	// Increment component byte offset
	offset := offset + SIZEOF(ST_RTComponentData) + qrtComponent[comp].nSize;
END_FOR

// Get hook position
IF bActive THEN
	IF markerComponent.nMarkers >= 2 THEN
		// Reset eMin to a default "high" value
		eMin := 1E10;
		
		FOR i := 0 TO markerComponent.nMarkers DO
			FOR j := 0 TO markerComponent.nMarkers DO
				// Calculate norm
				d := GetNorm(markerComponent.markers[i], markerComponent.markers[j]);
				e := ABS(d - dMarker);
				
				// Check if current marker set is closer than the others
				IF e < eMin THEN
					eMin := e;
					
					dSave := d;
					iSave := i;
					jSave := j;
				END_IF
			END_FOR
		END_FOR
		// Pick saved markers
		iMarker := markerComponent.markers[iSave];
		jMarker := markerComponent.markers[jSave];
		
		// Calculate average marker
		feedback.dist := dSave/1000.0;
		
		xSave := (iMarker.x + jMarker.x)/2.0;
		ySave := (iMarker.y + jMarker.y)/2.0;
		zSave := (iMarker.z + jMarker.z)/2.0;
		
	ELSIF markerComponent.nMarkers = 1 THEN
		// Indicate that hook is based on a single marker
		feedback.dist := 0.0;
		
		xSave := markerComponent.markers[0].x;
		ySave := markerComponent.markers[0].y;
		zSave := markerComponent.markers[0].z;
	ELSE	
		// Indicate that no markers are detected
		feedback.dist := -1.0;
	END_IF
	
	// mm -> m
	feedback.pos[0] := REAL_TO_LREAL(xSave/1000.0);
	feedback.pos[1] := REAL_TO_LREAL(ySave/1000.0);
	feedback.pos[2] := REAL_TO_LREAL(zSave/1000.0);
	
END_IF

METHOD FB_exit : BOOL
VAR_INPUT
	bInCopyCode : BOOL; // if TRUE, the exit method is called for exiting an instance that is copied afterwards (online change).
END_VAR
END_METHOD

METHOD FB_init : BOOL
VAR_INPUT
	bInitRetains : BOOL; // if TRUE, the retain variables are initialized (warm start / cold start)
	bInCopyCode : BOOL;  // if TRUE, the instance afterwards gets moved into the copy code (online change)

	// Init variables
	_localPort : UINT;
	_pTxHmi : POINTER TO ST_TxHmiQualisys;
END_VAR
// Initilize the udpServer
udpServer.FB_init(
	bInitRetains,
	bInCopyCode,
	_localPort,
	0,
	0,
	0,
	0
);

pTxHmi := _pTxHmi;
END_METHOD

METHOD FB_reinit : BOOL
VAR_INPUT
END_VAR
END_METHOD

METHOD PRIVATE GetNorm : REAL
VAR_INPUT
	m1 : ST_3DMarkerPositionNoLabel;
	m2 : ST_3DMarkerPositionNoLabel;
END_VAR

VAR
	x : REAL;
	y : REAL;
	z : REAL;
END_VAR
// Vector 
x := m2.x - m1.x;
y := m2.y - m1.y;
z := m2.z - m1.z;

// Norm
GetNorm := SQRT(x*x + y*y + z*z);
END_METHOD

METHOD PRIVATE UpdateHMI : BOOL
VAR_INPUT
END_VAR

VAR
	i : UDINT;
END_VAR
// Update global Hmi data
IF bActive THEN
	pTxHmi^.status := 0;
ELSE
	pTxHmi^.status := -1;
END_IF

// Update feedback data
pTxHmi^.dist := LREAL_TO_REAL(feedback.dist);
pTxHmi^.x := LREAL_TO_REAL(feedback.pos[0]);
pTxHmi^.y := LREAL_TO_REAL(feedback.pos[1]);
pTxHmi^.z := LREAL_TO_REAL(feedback.pos[2]);

// Marker data
FOR i := 0 TO 9 DO
	pTxHmi^.markers[i] := markerComponent.markers[i];
END_FOR
END_METHOD

END_FUNCTION_BLOCK

// ---- POUs/Interfaces/FB_LeicaInterface.TcPOU
FUNCTION_BLOCK FB_LeicaInterface
VAR_INPUT
END_VAR
VAR_OUTPUT
	feedback : ST_FeedbackLeica;
	active : BOOL := FALSE;
END_VAR
VAR
	// Variables linked to LeicaAT960 Box 1
	Status AT %I* : UDINT := 0;
	TimeStamp AT %I* : ULINT := 0;
	AngleHz AT %I* : LREAL := 0.0;
	AngleVt	AT %I* : LREAL := 0.0;
	Distance AT %I* : LREAL := 0.0;
	Quaternion0	AT %I* : LREAL := 1.0;
	Quaternion1	AT %I* : LREAL := 0.0;
	Quaternion2	AT %I* : LREAL := 0.0;
	Quaternion3	AT %I* : LREAL := 0.0;
	
	// Rotation matrix
	fbQuatToRotMatrix : FB_QuatToRotMatrix;
	rot : ARRAY [0..8] OF LREAL;
	
	// Actviity monitoring
	frame : ULINT := 0;
	frameOld : ULINT := 0;
	frameLoss : ULINT := 0;
END_VAR

// Check activity
frame := TimeStamp;
IF frame <> frameOld THEN
	// Update frame old
	frameOld := frame;
	
	// Reset frameLoss
	frameLoss := 0;
ELSE
	// Count frame losses
	frameLoss := frameLoss + 1;
END_IF

// Set activity status after 1 second given 5ms in ms
IF frameLoss > 200 THEN
	active := FALSE;
ELSE
	active := TRUE;
END_IF

// Leica transform to x, y and z coordinates
feedback.pos[0] := Distance*SIN(AngleVt)*SIN(AngleHz);
feedback.pos[1] := Distance*SIN(AngleVt)*COS(AngleHz);
feedback.pos[2] := Distance*COS(AngleVt);

// Convert to rotation matrix
fbQuatToRotMatrix(
	w := Quaternion0,
	x := Quaternion1,
	y := Quaternion2,
	z := Quaternion3
);

feedback.R11 := fbQuatToRotMatrix.R11;
feedback.R12 := fbQuatToRotMatrix.R12;
feedback.R13 := fbQuatToRotMatrix.R13;

feedback.R21 := fbQuatToRotMatrix.R21;
feedback.R22 := fbQuatToRotMatrix.R22;
feedback.R23 := fbQuatToRotMatrix.R23;

feedback.R31 := fbQuatToRotMatrix.R31;
feedback.R32 := fbQuatToRotMatrix.R32;
feedback.R33 := fbQuatToRotMatrix.R33;

END_FUNCTION_BLOCK

// ---- POUs/Simulink/FB_QuatToRotMatrix.TcPOU
FUNCTION_BLOCK FB_QuatToRotMatrix
VAR_INPUT
	w: LREAL := 1.0;
	x: LREAL := 0.0;
	y: LREAL := 0.0;
	z: LREAL := 0.0;
END_VAR
VAR_OUTPUT
	R11: LREAL;
	R12: LREAL;
	R13: LREAL;
	R21: LREAL;
	R22: LREAL;
	R23: LREAL;
	R31: LREAL;
	R32: LREAL;
	R33: LREAL;
END_VAR
VAR
	b_R: ARRAY[0..8] OF LREAL;
	tempR: ARRAY[0..8] OF LREAL;
	y_0: LREAL;
	outsz: ARRAY[0..2] OF SINT;
	iwork: ARRAY[0..2] OF DINT;
	idest: DINT;
	isrc: DINT;
	normRowMatrix_idx_0: LREAL;
	normRowMatrix_idx_2: LREAL;
	normRowMatrix_idx_1: LREAL;
	tempR_tmp: LREAL;
	tempR_tmp_0: LREAL;
	tempR_tmp_1: LREAL;
	tempR_tmp_2: LREAL;
	tempR_tmp_3: LREAL;
	tempR_tmp_4: LREAL;
	exitg1: DINT;
END_VAR


(* MATLAB Function: '<Root>/FB_QuatToRotMatrix' *)
(* MATLAB Function 'FB_QuatToRotMatrix': '<S1>:1' *)
(* '<S1>:1:3' quat = [w, x, y, z]; *)
(* '<S1>:1:5' R = quat2rotm(quat); *)
y_0 := 1.0 / SQRT((((w * w) + (x * x)) + (y * y)) + (z * z));
normRowMatrix_idx_0 := w * y_0;
normRowMatrix_idx_1 := x * y_0;
normRowMatrix_idx_2 := y * y_0;
y_0 := z * y_0;
tempR_tmp_1 := y_0 * y_0;
tempR_tmp_4 := normRowMatrix_idx_2 * normRowMatrix_idx_2;
tempR[0] := 1.0 - ((tempR_tmp_4 + tempR_tmp_1) * 2.0);
tempR_tmp := normRowMatrix_idx_1 * normRowMatrix_idx_2;
tempR_tmp_0 := normRowMatrix_idx_0 * y_0;
tempR[1] := (tempR_tmp - tempR_tmp_0) * 2.0;
tempR_tmp_2 := normRowMatrix_idx_1 * y_0;
tempR_tmp_3 := normRowMatrix_idx_0 * normRowMatrix_idx_2;
tempR[2] := (tempR_tmp_2 + tempR_tmp_3) * 2.0;
tempR[3] := (tempR_tmp + tempR_tmp_0) * 2.0;
tempR_tmp := normRowMatrix_idx_1 * normRowMatrix_idx_1;
tempR[4] := 1.0 - ((tempR_tmp + tempR_tmp_1) * 2.0);
tempR_tmp_1 := normRowMatrix_idx_2 * y_0;
tempR_tmp_0 := normRowMatrix_idx_0 * normRowMatrix_idx_1;
tempR[5] := (tempR_tmp_1 - tempR_tmp_0) * 2.0;
tempR[6] := (tempR_tmp_2 - tempR_tmp_3) * 2.0;
tempR[7] := (tempR_tmp_1 + tempR_tmp_0) * 2.0;
tempR[8] := 1.0 - ((tempR_tmp + tempR_tmp_4) * 2.0);
outsz[0] := 3;
outsz[1] := 3;
outsz[2] := 1;
iwork[0] := 0;
iwork[1] := 0;
iwork[2] := 0;
idest := 0;
REPEAT 
    isrc := (iwork[2] * 3) + iwork[1];
    b_R[idest] := tempR[isrc];
    idest := idest + 1;
    isrc := isrc + 3;
    b_R[idest] := tempR[isrc];
    idest := idest + 1;
    isrc := isrc + 3;
    b_R[idest] := tempR[isrc];
    idest := idest + 1;
    isrc := 1;
    REPEAT 
        exitg1 := 0;
        iwork[isrc] := iwork[isrc] + 1;

        IF iwork[isrc] < SINT_TO_DINT(outsz[isrc]) THEN 
            exitg1 := 2;
        ELSIF (isrc + 1) = 3 THEN 
            exitg1 := 1;
        ELSE 
            iwork[1] := 0;
            isrc := 2;
        END_IF;

    UNTIL NOT(exitg1 = 0)
    END_REPEAT;
UNTIL NOT( NOT (exitg1 = 1))
END_REPEAT;
(* Outport: '<Root>/R11' incorporates:
 *  MATLAB Function: '<Root>/FB_QuatToRotMatrix' *)
(* '<S1>:1:7' R11 = R(1,1); *)
(* '<S1>:1:8' R12 = R(1,2); *)
(* '<S1>:1:9' R13 = R(1,3); *)
(* '<S1>:1:11' R21 = R(2,1); *)
(* '<S1>:1:12' R22 = R(2,2); *)
(* '<S1>:1:13' R23 = R(2,3); *)
(* '<S1>:1:15' R31 = R(3,1); *)
(* '<S1>:1:16' R32 = R(3,2); *)
(* '<S1>:1:17' R33 = R(3,3); *)
R11 := b_R[0];
(* Outport: '<Root>/R12' incorporates:
 *  MATLAB Function: '<Root>/FB_QuatToRotMatrix' *)
R12 := b_R[3];
(* Outport: '<Root>/R13' incorporates:
 *  MATLAB Function: '<Root>/FB_QuatToRotMatrix' *)
R13 := b_R[6];
(* Outport: '<Root>/R21' incorporates:
 *  MATLAB Function: '<Root>/FB_QuatToRotMatrix' *)
R21 := b_R[1];
(* Outport: '<Root>/R22' incorporates:
 *  MATLAB Function: '<Root>/FB_QuatToRotMatrix' *)
R22 := b_R[4];
(* Outport: '<Root>/R23' incorporates:
 *  MATLAB Function: '<Root>/FB_QuatToRotMatrix' *)
R23 := b_R[7];
(* Outport: '<Root>/R31' incorporates:
 *  MATLAB Function: '<Root>/FB_QuatToRotMatrix' *)
R31 := b_R[2];
(* Outport: '<Root>/R32' incorporates:
 *  MATLAB Function: '<Root>/FB_QuatToRotMatrix' *)
R32 := b_R[5];
(* Outport: '<Root>/R33' incorporates:
 *  MATLAB Function: '<Root>/FB_QuatToRotMatrix' *)
R33 := b_R[8];

END_FUNCTION_BLOCK

// ---- POUs/CSV/FB_CsvReader.TcPOU
FUNCTION_BLOCK FB_CsvReader
VAR_INPUT
	bStart : BOOL;
	
END_VAR
VAR_OUTPUT
	data : ARRAY [0..100] OF T_MaxString;
END_VAR

VAR
	sNetId : T_MaxString := '';
	bOpen : BOOL;
	bClose : BOOL;
	
	fbOpen : FB_FileOpen;
	fbClose : FB_FileClose;
	
	fbWriter : FB_CSVMemBufferWriter;
	
	n : UDINT;
	i : UDINT;

	
	
	
	eState : INT;
END_VAR

n := n + 1;
CASE eState OF
	-1 : // ERROR
			
	
	0 : // Idle
		i := 0;
	
	1 : // Start open
		fbOpen(
			sNetId := sNetId,
			sPathName := 'C:\test.txt',
			nMode := FOPEN_MODEWRITE OR FOPEN_MODETEXT,
			ePath := PATH_GENERIC,
			bExecute := TRUE
		);
		
		eState := 2;
	
	2 : // Open
		fbOpen(bExecute := FALSE);
		
		IF NOT fbOpen.bBusy THEN
			IF NOT fbOpen.bError THEN
				eState := 3;
				
			ELSE
				eState := - 1;
				
			END_IF
		END_IF
		
	3 : // File redy

		IF bStart THEN
			eState := 4;
			
		END_IF;
		
	4 : // Start to record data to CSV file
	
		
	
	
	100 : // Start close
		fbClose(
			sNetId := sNetId,
			hFile := fbOpen.hFile,
			bExecute := TRUE
		);
		
		eState := 101;
		
	101: // Close
		fbClose(bExecute := FALSE);
		
		IF NOT fbClose.bBusy THEN
			IF NOT fbClose.bError THEN
				eState := 0;
				
			ELSE
				eState := -1;
				
			END_IF
			
		END_IF
		
	
END_CASE

END_FUNCTION_BLOCK

// ---- POUs/Utils/F_VelocityBoundary.TcPOU
FUNCTION F_VelocityBoundary : ARRAY [0..1] OF LREAL;
VAR_INPUT
	q : LREAL; // Current position
	qMin : LREAL; // Min position
	qMax : LREAL; // Max position
	V : LREAL := 0.1; // Max allowed velocity
	A : LREAL := 1; // max allowed acceleration
	Ts : LREAL := 0.005; // Task time step
	
END_VAR
VAR
	qMin_t : LREAL;
	qMax_t : LREAL;
	
	t0, t1, t2 : LREAL; 
	
END_VAR

// Ensure Ts is positive
Ts := ABS(Ts); 

// Ensure that V and A is positive
V := ABS(V);
A := ABS(A);

// Ensure q is in [qMin, qMax]
q := MAX(q, qMin);
q := MIN(q, qMax);

// Lower Boundary       
t0 := (qMin - q)/Ts;
t1 := -V;
t2 := -SQRT(ABS(2*A*(q - qMin)));

qMin_t := MAX(t0, MAX(t1, t2));

// Upper Boundary
t0 := (qMax - q)/Ts;
t1 := V;
t2 := SQRT(ABS(2*A*(qMax - q)));

qMax_t := MIN(t0, MIN(t1, t2));

// Return velocity bound
F_VelocityBoundary[0] := qMin_t;
F_VelocityBoundary[1] := qMax_t;

END_FUNCTION

// ---- SystemFunctions/CheckDivReal.TcPOU
FUNCTION CheckDivReal  : REAL
VAR_INPUT
	divisor : REAL;
END_VAR
VAR
END_VAR

IF divisor = 0 THEN
        CheckDivReal := 1E-10;
ELSE
        CheckDivReal := divisor;
END_IF

END_FUNCTION

// ---- SystemFunctions/CheckDivLReal.TcPOU
FUNCTION CheckDivLReal  : LREAL
VAR_INPUT
	divisor : LREAL;
END_VAR
VAR
END_VAR

IF divisor = 0 THEN
        CheckDivReal := 1E-10;
ELSE
        CheckDivReal := divisor;
END_IF

END_FUNCTION
